FUNCTION_BLOCK AGENT_RECV (* Composite Function Block Type *)
  (* Standard: 61499-2 *)
  (* Version 1.0, 2019-11-11, badger *)
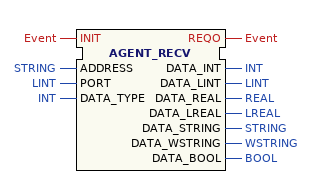
  EVENT_INPUT
    INIT; (* Initialization Request *)
  END_EVENT
  EVENT_OUTPUT
    REQO;
  END_EVENT
  VAR_INPUT
    ADDRESS : STRING;
    PORT : LINT;
    DATA_TYPE : INT;
  END_VAR
  VAR_OUTPUT
    DATA_INT : INT;
    DATA_LINT : LINT;
    DATA_REAL : REAL;
    DATA_LREAL : LREAL;
    DATA_STRING : STRING;
    DATA_WSTRING : WSTRING;
    DATA_BOOL : BOOL;
  END_VAR
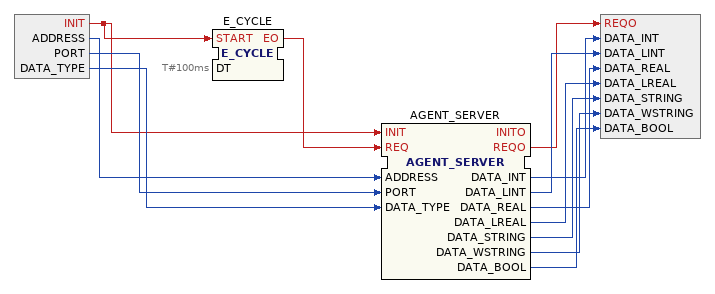
  FBS
    E_CYCLE : E_CYCLE(DT := T#100ms);
    AGENT_SERVER : AGENT_SERVER;
  END_FBS
  EVENT_CONNECTIONS
    INIT TO E_CYCLE.START;
    INIT TO AGENT_SERVER.INIT;
    E_CYCLE.EO TO AGENT_SERVER.REQ;
    AGENT_SERVER.REQO TO REQO;
  END_CONNECTIONS
  DATA_CONNECTIONS
    ADDRESS TO AGENT_SERVER.ADDRESS;
    PORT TO AGENT_SERVER.PORT;
    DATA_TYPE TO AGENT_SERVER.DATA_TYPE;
    AGENT_SERVER.DATA_INT TO DATA_INT;
    AGENT_SERVER.DATA_LINT TO DATA_LINT;
    AGENT_SERVER.DATA_REAL TO DATA_REAL;
    AGENT_SERVER.DATA_LREAL TO DATA_LREAL;
    AGENT_SERVER.DATA_STRING TO DATA_STRING;
    AGENT_SERVER.DATA_WSTRING TO DATA_WSTRING;
    AGENT_SERVER.DATA_BOOL TO DATA_BOOL;
  END_CONNECTIONS
END_FUNCTION_BLOCK
